LIN {X 0,Y 115.59,Z 711.815,A -85,B 0,C 180,E1 -30048.636,E2 -30048.636} C_VEL
LIN {X 0,Y 121.529,Z 700.022,A -85,B 0,C 180,E1 -30049.447,E2 -30049.447} C_VEL
LIN {X 0,Y 126.039,Z 688.294,A -85,B 0,C 180,E1 -30050.037,E2 -30050.037} C_VEL
LIN {X 0,Y 129.547,Z 675.475,A -85,B 0,C 180,E1 -30050.461,E2 -30050.461} C_VEL
LIN {X 0,Y 131.84,Z 661.062,A -85,B 0,C 180,E1 -30050.822,E2 -30050.822} C_VEL
LIN {X 0,Y 132.217,Z 657.756,A -85,B 0,C 180,E1 -30050.921,E2 -30050.921} C_VEL
LIN {X 0,Y 131.722,Z 655.629,A -85,B 0,C 180,E1 -30053.683,E2 -30053.683} C_VEL
LIN {X 0,Y 131.497,Z 654.069,A -85,B 0,C 180,E1 -30056.17,E2 -30056.17} C_VEL
LIN {X 0,Y 131.404,Z 653.558,A -85,B 0,C 180,E1 -30060.001,E2 -30060.001} C_VEL
LIN {X 0,Y 131.546,Z 654.495,A -85,B 0,C 180,E1 -30062.788,E2 -30062.788} C_VEL
LIN {X 0,Y 131.537,Z 656.009,A -85,B 0,C 180,E1 -30063.787,E2 -30063.787} C_VEL
LIN {X 0,Y 131.334,Z 659.04,A -85,B 0,C 180,E1 -30064.554,E2 -30064.554} C_VEL
LIN {X 0,Y 130.805,Z 663.674,A -85,B 0,C 180,E1 -30064.929,E2 -30064.929} C_VEL
LIN {X 0,Y 129.936,Z 669.022,A -85,B 0,C 180,E1 -30064.793,E2 -30064.793} C_VEL
LIN {X 0,Y 128.707,Z 675.107,A -85,B 0,C 180,E1 -30064.796,E2 -30064.796} C_VEL
LIN {X 0,Y 125.026,Z 688.126,A -85,B 0,C 180,E1 -30065.242,E2 -30065.242} C_VEL
LIN {X 0,Y 120.094,Z 700.491,A -85,B 0,C 180,E1 -30065.831,E2 -30065.831} C_VEL
LIN {X 0,Y 114.09,Z 711.929,A -85,B 0,C 180,E1 -30066.646,E2 -30066.646} C_VEL
LIN {X 0,Y 106.425,Z 723.397,A -85,B 0,C 180,E1 -30067.891,E2 -30067.891} C_VEL
LIN {X 0,Y 97.926,Z 733.578,A -85,B 0,C 180,E1 -30069.321,E2 -30069.321} C_VEL
LIN {X 0,Y 89.47,Z 741.809,A -85,B 0,C 180,E1 -30070.928,E2 -30070.928} C_VEL
LIN {X 0,Y 79.475,Z 749.839,A -85,B 0,C 180,E1 -30073.417,E2 -30073.417} C_VEL
LIN {X 0,Y 69.638,Z 756.292,A -85,B 0,C 180,E1 -30076.516,E2 -30076.516} C_VEL
LIN {X 0,Y 60.109,Z 761.402,A -85,B 0,C 180,E1 -30080.716,E2 -30080.716} C_VEL
LIN {X 0,Y 51.033,Z 765.333,A -85,B 0,C 180,E1 -30086.475,E2 -30086.475} C_VEL
LIN {X 0,Y 42.512,Z 768.222,A -85,B 0,C 180,E1 -30094.253,E2 -30094.253} C_VEL
LIN {X 0,Y 33.116,Z 770.553,A -85,B 0,C 180,E1 -30110.457,E2 -30110.457} C_VEL
LIN {X 0,Y 29.749,Z 771.131,A -85,B 0,C 180,E1 -30121.805,E2 -30121.805} C_VEL
LIN {X 0,Y 27.663,Z 771.312,A -85,B 0,C 180,E1 -30135.283,E2 -30135.283} C_VEL
LIN {X 0,Y 27.148,Z 771.065,A -85,B 0,C 180,E1 -30150,E2 -30150} C_VEL
LIN {X 0,Y 28.19,Z 770.44,A -85,B 0,C 180,E1 -30164.436,E2 -30164.436} C_VEL
LIN {X 0,Y 30.59,Z 769.436,A -85,B 0,C 180,E1 -30177.354,E2 -30177.354} C_VEL
LIN {X 0,Y 34.116,Z 768.006,A -85,B 0,C 180,E1 -30188.17,E2 -30188.17} C_VEL
LIN {X 0,Y 41.107,Z 765.059,A -85,B 0,C 180,E1 -30200.294,E2 -30200.294} C_VEL
LIN {X 0,Y 46.719,Z 762.376,A -85,B 0,C 180,E1 -30206.52,E2 -30206.52} C_VEL
LIN {X 0,Y 46.259,Z 762.112,A -85,B 0,C 180,E1 -30209.388,E2 -30209.388} C_VEL
LIN {X 0,Y 44.988,Z 762.224,A -85,B 0,C 180,E1 -30212.05,E2 -30212.05} C_VEL
LIN {X 0,Y 42.91,Z 762.139,A -85,B 0,C 180,E1 -30220.876,E2 -30220.876} C_VEL
LIN {X 0,Y 41.474,Z 762.242,A -85,B 0,C 180,E1 -30230.242,E2 -30230.242} C_VEL
LIN {X 0,Y 45.335,Z 762.004,A -85,B 0,C 180,E1 -30258.06,E2 -30258.06} C_VEL
LIN {X 0,Y 48.651,Z 761.909,A -85,B 0,C 180,E1 -30265.68,E2 -30265.68} C_VEL
LIN {X 0,Y 47.899,Z 762.718,A -85,B 0,C 180,E1 -30268.318,E2 -30268.318} C_VEL
LIN {X 0,Y 39.67,Z 766.691,A -85,B 0,C 180,E1 -30277.135,E2 -30277.135} C_VEL
LIN {X 0,Y 32.833,Z 769.618,A -85,B 0,C 180,E1 -30290.048,E2 -30290.048} C_VEL
LIN {X 0,Y 29.517,Z 771.007,A -85,B 0,C 180,E1 -30301.563,E2 -30301.563} C_VEL
LIN {X 0,Y 27.544,Z 771.994,A -85,B 0,C 180,E1 -30315.217,E2 -30315.217} C_VEL
LIN {X 0,Y 27.126,Z 772.588,A -85,B 0,C 180,E1 -30330,E2 -30330} C_VEL
LIN {X 0,Y 27.557,Z 772.746,A -85,B 0,C 180,E1 -30344.775,E2 -30344.775} C_VEL
LIN {X 0,Y 32.899,Z 771.821,A -85,B 0,C 180,E1 -30369.856,E2 -30369.856} C_VEL
LIN {X 0,Y 37.238,Z 770.778,A -85,B 0,C 180,E1 -30379.017,E2 -30379.017} C_VEL
LIN {X 0,Y 42.388,Z 769.299,A -85,B 0,C 180,E1 -30385.996,E2 -30385.996} C_VEL
LIN {X 0,Y 50.941,Z 766.283,A -85,B 0,C 180,E1 -30393.733,E2 -30393.733} C_VEL
LIN {X 0,Y 62.114,Z 761.207,A -85,B 0,C 180,E1 -30400.159,E2 -30400.159} C_VEL
LIN {X 0,Y 72.994,Z 754.959,A -85,B 0,C 180,E1 -30404.322,E2 -30404.322} C_VEL
LIN {X 0,Y 82.933,Z 747.864,A -85,B 0,C 180,E1 -30407.037,E2 -30407.037} C_VEL
LIN {X 0,Y 93.039,Z 739.053,A -85,B 0,C 180,E1 -30409.105,E2 -30409.105} C_VEL
LIN {X 0,Y 101.542,Z 729.994,A -85,B 0,C 180,E1 -30410.49,E2 -30410.49} C_VEL
LIN {X 0,Y 109.243,Z 719.912,A -85,B 0,C 180,E1 -30411.535,E2 -30411.535} C_VEL
LIN {X 0,Y 116.123,Z 708.762,A -85,B 0,C 180,E1 -30412.319,E2 -30412.319} C_VEL
LIN {X 0,Y 121.57,Z 697.557,A -85,B 0,C 180,E1 -30412.908,E2 -30412.908} C_VEL
LIN {X 0,Y 126.04,Z 685.303,A -85,B 0,C 180,E1 -30413.325,E2 -30413.325} C_VEL
LIN {X 0,Y 129.305,Z 672.284,A -85,B 0,C 180,E1 -30413.636,E2 -30413.636} C_VEL
LIN {X 0,Y 130.784,Z 662.762,A -85,B 0,C 180,E1 -30413.928,E2 -30413.928} C_VEL
LIN {X 0,Y 130.572,Z 660.969,A -85,B 0,C 180,E1 -30416.915,E2 -30416.915} C_VEL
LIN {X 0,Y 130.533,Z 660.648,A -85,B 0,C 180,E1 -30420.001,E2 -30420.001} C_VEL
LIN {X 0,Y 130.622,Z 661.461,A -85,B 0,C 180,E1 -30422.313,E2 -30422.313} C_VEL
LIN {X 0,Y 130.818,Z 662.851,A -85,B 0,C 180,E1 -30424.506,E2 -30424.506} C_VEL
LIN {X 0,Y 128.707,Z 675.107,A -85,B 0,C 180,E1 -30424.796,E2 -30424.796} C_VEL
LIN {X 0,Y 127.276,Z 680.841,A -85,B 0,C 180,E1 -30424.597,E2 -30424.597} C_VEL
LIN {X 0,Y 124.145,Z 690.015,A -85,B 0,C 180,E1 -30423.615,E2 -30423.615} C_VEL
LIN {X 0,Y 120.303,Z 698.922,A -85,B 0,C 180,E1 -30422.7,E2 -30422.7} C_VEL
LIN {X 0,Y 117.718,Z 704.215,A -85,B 0,C 180,E1 -30422.644,E2 -30422.644} C_VEL
LIN {X 0,Y 111.05,Z 715.823,A -85,B 0,C 180,E1 -30423.361,E2 -30423.361} C_VEL
LIN {X 0,Y 103.089,Z 726.716,A -85,B 0,C 180,E1 -30424.425,E2 -30424.425} C_VEL
LIN {X 0,Y 93.572,Z 737.144,A -85,B 0,C 180,E1 -30425.641,E2 -30425.641} C_VEL
LIN {X 0,Y 84.967,Z 744.801,A -85,B 0,C 180,E1 -30426.999,E2 -30426.999} C_VEL
LIN {X 0,Y 74.727,Z 752.258,A -85,B 0,C 180,E1 -30429.071,E2 -30429.071} C_VEL
LIN {X 0,Y 64.603,Z 758.242,A -85,B 0,C 180,E1 -30431.743,E2 -30431.743} C_VEL
LIN {X 0,Y 54.708,Z 762.953,A -85,B 0,C 180,E1 -30435.539,E2 -30435.539} C_VEL
LIN {X 0,Y 45.124,Z 766.538,A -85,B 0,C 180,E1 -30440.857,E2 -30440.857} C_VEL
LIN {X 0,Y 38.955,Z 768.384,A -85,B 0,C 180,E1 -30445.573,E2 -30445.573} C_VEL
LIN {X 0,Y 33.169,Z 769.762,A -85,B 0,C 180,E1 -30452.056,E2 -30452.056} C_VEL
LIN {X 0,Y 23.716,Z 771.314,A -85,B 0,C 180,E1 -30473.654,E2 -30473.654} C_VEL
LIN {X 0,Y 20.883,Z 771.504,A -85,B 0,C 180,E1 -30490.335,E2 -30490.335} C_VEL
LIN {X 0,Y 20.042,Z 771.264,A -85,B 0,C 180,E1 -30510,E2 -30510} C_VEL
LIN {X 0,Y 21.406,Z 770.644,A -85,B 0,C 180,E1 -30529.166,E2 -30529.166} C_VEL
LIN {X 0,Y 24.5,Z 769.646,A -85,B 0,C 180,E1 -30545.008,E2 -30545.008} C_VEL
LIN {X 0,Y 28.875,Z 768.227,A -85,B 0,C 180,E1 -30556.899,E2 -30556.899} C_VEL
LIN {X 0,Y 38.008,Z 764.859,A -85,B 0,C 180,E1 -30569.88,E2 -30569.88} C_VEL
LIN {X 0,Y 37.473,Z 764.693,A -85,B 0,C 180,E1 -30573.661,E2 -30573.661} C_VEL
LIN {X 0,Y 36.261,Z 764.773,A -85,B 0,C 180,E1 -30611.173,E2 -30611.173} C_VEL
LIN {X 0,Y 39.092,Z 764.687,A -85,B 0,C 180,E1 -30621.071,E2 -30621.071} C_VEL
LIN {X 0,Y 38.792,Z 765.232,A -85,B 0,C 180,E1 -30625.063,E2 -30625.063} C_VEL
LIN {X 0,Y 32.944,Z 767.529,A -85,B 0,C 180,E1 -30631.427,E2 -30631.427} C_VEL
LIN {X 0,Y 27.745,Z 769.399,A -85,B 0,C 180,E1 -30640.545,E2 -30640.545} C_VEL
LIN {X 0,Y 23.494,Z 770.797,A -85,B 0,C 180,E1 -30653.254,E2 -30653.254} C_VEL
LIN {X 0,Y 20.748,Z 771.789,A -85,B 0,C 180,E1 -30670.201,E2 -30670.201} C_VEL
LIN {X 0,Y 20.018,Z 772.388,A -85,B 0,C 180,E1 -30690,E2 -30690} C_VEL
LIN {X 0,Y 20.761,Z 772.557,A -85,B 0,C 180,E1 -30709.786,E2 -30709.786} C_VEL
LIN {X 0,Y 27.799,Z 771.643,A -85,B 0,C 180,E1 -30739.325,E2 -30739.325} C_VEL
LIN {X 0,Y 33.001,Z 770.606,A -85,B 0,C 180,E1 -30748.411,E2 -30748.411} C_VEL
LIN {X 0,Y 38.851,Z 769.138,A -85,B 0,C 180,E1 -30754.751,E2 -30754.751} C_VEL
LIN {X 0,Y 48.215,Z 766.135,A -85,B 0,C 180,E1 -30761.342,E2 -30761.342} C_VEL
LIN {X 0,Y 59.314,Z 761.438,A -85,B 0,C 180,E1 -30766.293,E2 -30766.293} C_VEL
LIN {X 0,Y 71.402,Z 754.842,A -85,B 0,C 180,E1 -30769.822,E2 -30769.822} C_VEL
LIN {X 0,Y 81.635,Z 747.768,A -85,B 0,C 180,E1 -30771.899,E2 -30771.899} C_VEL
LIN {X 0,Y 91.96,Z 738.978,A -85,B 0,C 180,E1 -30773.46,E2 -30773.46} C_VEL
LIN {X 0,Y 100.611,Z 729.948,A -85,B 0,C 180,E1 -30774.494,E2 -30774.494} C_VEL
LIN {X 0,Y 108.427,Z 719.906,A -85,B 0,C 180,E1 -30775.239,E2 -30775.239} C_VEL
LIN {X 0,Y 115.389,Z 708.8,A -85,B 0,C 180,E1 -30775.81,E2 -30775.81} C_VEL
LIN {X 0,Y 121.282,Z 696.784,A -85,B 0,C 180,E1 -30776.264,E2 -30776.264} C_VEL
LIN {X 0,Y 125.89,Z 683.969,A -85,B 0,C 180,E1 -30776.556,E2 -30776.556} C_VEL
LIN {X 0,Y 129.144,Z 670.629,A -85,B 0,C 180,E1 -30776.816,E2 -30776.816} C_VEL
LIN {X 0,Y 129.549,Z 668.159,A -85,B 0,C 180,E1 -30776.891,E2 -30776.891} C_VEL
LIN {X 0,Y 129.532,Z 667.718,A -85,B 0,C 180,E1 -30780.001,E2 -30780.001} C_VEL
LIN {X 0,Y 129.541,Z 668.233,A -85,B 0,C 180,E1 -30781.471,E2 -30781.471} C_VEL
LIN {X 0,Y 126.782,Z 680.85,A -85,B 0,C 180,E1 -30781.786,E2 -30781.786} C_VEL
LIN {X 0,Y 122.426,Z 693.772,A -85,B 0,C 180,E1 -30782.194,E2 -30782.194} C_VEL
LIN {X 0,Y 117.718,Z 704.215,A -85,B 0,C 180,E1 -30782.644,E2 -30782.644} C_VEL
LIN {X 0,Y 114.915,Z 709.418,A -85,B 0,C 180,E1 -30782.615,E2 -30782.615} C_VEL
LIN {X 0,Y 109.743,Z 717.691,A -85,B 0,C 180,E1 -30781.745,E2 -30781.745} C_VEL
LIN {X 0,Y 103.924,Z 725.496,A -85,B 0,C 180,E1 -30780.792,E2 -30780.792} C_VEL
LIN {X 0,Y 100.069,Z 729.966,A -85,B 0,C 180,E1 -30780.712,E2 -30780.712} C_VEL
LIN {X 0,Y 91.391,Z 738.842,A -85,B 0,C 180,E1 -30781.447,E2 -30781.447} C_VEL
LIN {X 0,Y 80.906,Z 747.563,A -85,B 0,C 180,E1 -30782.642,E2 -30782.642} C_VEL
LIN {X 0,Y 70.463,Z 754.546,A -85,B 0,C 180,E1 -30784.151,E2 -30784.151} C_VEL
LIN {X 0,Y 60.091,Z 760.088,A -85,B 0,C 180,E1 -30786.227,E2 -30786.227} C_VEL
LIN {X 0,Y 49.838,Z 764.419,A -85,B 0,C 180,E1 -30789.213,E2 -30789.213} C_VEL
LIN {X 0,Y 43.106,Z 766.693,A -85,B 0,C 180,E1 -30791.978,E2 -30791.978} C_VEL
LIN {X 0,Y 36.455,Z 768.545,A -85,B 0,C 180,E1 -30795.443,E2 -30795.443} C_VEL
LIN {X 0,Y 29.997,Z 769.934,A -85,B 0,C 180,E1 -30800.424,E2 -30800.424} C_VEL
LIN {X 0,Y 18.478,Z 771.497,A -85,B 0,C 180,E1 -30820.475,E2 -30820.475} C_VEL
LIN {X 0,Y 14.389,Z 771.696,A -85,B 0,C 180,E1 -30840.764,E2 -30840.764} C_VEL
LIN {X 0,Y 12.951,Z 771.463,A -85,B 0,C 180,E1 -30870,E2 -30870} C_VEL
LIN {X 0,Y 14.894,Z 770.848,A -85,B 0,C 180,E1 -30898.154,E2 -30898.154} C_VEL
LIN {X 0,Y 19.128,Z 769.856,A -85,B 0,C 180,E1 -30917.293,E2 -30917.293} C_VEL
LIN {X 0,Y 28.63,Z 767.264,A -85,B 0,C 180,E1 -30934.382,E2 -30934.382} C_VEL
LIN {X 0,Y 29.039,Z 766.897,A -85,B 0,C 180,E1 -30940.375,E2 -30940.375} C_VEL
LIN {X 0,Y 29.672,Z 766.991,A -85,B 0,C 180,E1 -30973.698,E2 -30973.698} C_VEL
LIN {X 0,Y 29.855,Z 767.302,A -85,B 0,C 180,E1 -30979.678,E2 -30979.678} C_VEL
LIN {X 0,Y 23.727,Z 769.179,A -85,B 0,C 180,E1 -30987.304,E2 -30987.304} C_VEL
LIN {X 0,Y 18.291,Z 770.586,A -85,B 0,C 180,E1 -30999.787,E2 -30999.787} C_VEL
LIN {X 0,Y 14.25,Z 771.584,A -85,B 0,C 180,E1 -31020.451,E2 -31020.451} C_VEL
LIN {X 0,Y 12.924,Z 772.189,A -85,B 0,C 180,E1 -31050,E2 -31050} C_VEL
LIN {X 0,Y 14.262,Z 772.367,A -85,B 0,C 180,E1 -31079.523,E2 -31079.523} C_VEL
LIN {X 0,Y 23.766,Z 771.464,A -85,B 0,C 180,E1 -31112.513,E2 -31112.513} C_VEL
LIN {X 0,Y 29.889,Z 770.433,A -85,B 0,C 180,E1 -31120.137,E2 -31120.137} C_VEL
LIN {X 0,Y 36.386,Z 768.977,A -85,B 0,C 180,E1 -31124.958,E2 -31124.958} C_VEL
LIN {X 0,Y 46.431,Z 765.986,A -85,B 0,C 180,E1 -31129.689,E2 -31129.689} C_VEL
LIN {X 0,Y 57.084,Z 761.748,A -85,B 0,C 180,E1 -31132.93,E2 -31132.93} C_VEL
LIN {X 0,Y 68.755,Z 755.726,A -85,B 0,C 180,E1 -31135.272,E2 -31135.272} C_VEL
LIN {X 0,Y 79.194,Z 748.96,A -85,B 0,C 180,E1 -31136.706,E2 -31136.706} C_VEL
LIN {X 0,Y 89.675,Z 740.506,A -85,B 0,C 180,E1 -31137.728,E2 -31137.728} C_VEL
LIN {X 0,Y 98.427,Z 731.822,A -85,B 0,C 180,E1 -31138.418,E2 -31138.418} C_VEL
LIN {X 0,Y 107.192,Z 721.142,A -85,B 0,C 180,E1 -31138.946,E2 -31138.946} C_VEL
LIN {X 0,Y 112.456,Z 713.291,A -85,B 0,C 180,E1 -31139.225,E2 -31139.225} C_VEL
LIN {X 0,Y 112.449,Z 713.292,A -85,B 0,C 180,E1 -31139.556,E2 -31139.556} C_VEL
LIN {X 0,Y 104.54,Z 724.592,A -85,B 0,C 180,E1 -31140.29,E2 -31140.29} C_VEL
LIN {X 0,Y 100.069,Z 729.966,A -85,B 0,C 180,E1 -31140.712,E2 -31140.712} C_VEL
LIN {X 0,Y 99.544,Z 731.32,A -85,B 0,C 180,E1 -31140.746,E2 -31140.746} C_VEL
LIN {X 0,Y 99.544,Z 772.025,A -85,B 0,C 180,E1 -31140.746,E2 -31140.746} C_VEL
LIN {X 0,Y 59.705,Z 772.025,A -85,B 0,C 180,E1 -31139.693,E2 -31139.693} C_VEL
LIN {X 0,Y 57.707,Z 770.025,A -85,B 0,C 180,E1 -31139.602,E2 -31139.602} C_VEL
LIN {X 0,Y 57.707,Z 764.186,A -85,B 0,C 180,E1 -31139.602,E2 -31139.602} C_VEL
LIN {X 0,Y 55.003,Z 762.325,A -85,B 0,C 180,E1 -31140.002,E2 -31140.002} C_VEL
LIN {X 0,Y 42.205,Z 766.848,A -85,B 0,C 180,E1 -31142.448,E2 -31142.448} C_VEL
LIN {X 0,Y 35.235,Z 768.705,A -85,B 0,C 180,E1 -31144.236,E2 -31144.236} C_VEL
LIN {X 0,Y 28.308,Z 770.107,A -85,B 0,C 180,E1 -31146.765,E2 -31146.765} C_VEL
LIN {X 0,Y 14.873,Z 771.681,A -85,B 0,C 180,E1 -31159.083,E2 -31159.083} C_VEL
LIN {X 0,Y 8.898,Z 771.888,A -85,B 0,C 180,E1 -31177.834,E2 -31177.834} C_VEL
LIN {X 0,Y 5.87,Z 771.662,A -85,B 0,C 180,E1 -31230,E2 -31230} C_VEL
LIN {X 0,Y 9.262,Z 771.053,A -85,B 0,C 180,E1 -31279.355,E2 -31279.355} C_VEL
LIN {X 0,Y 20.134,Z 769.048,A -85,B 0,C 180,E1 -31303.714,E2 -31303.714} C_VEL
LIN {X 0,Y 21.237,Z 768.763,A -85,B 0,C 180,E1 -31313.11,E2 -31313.11} C_VEL
LIN {X 0,Y 21.34,Z 768.778,A -85,B 0,C 180,E1 -31319.996,E2 -31319.996} C_VEL
LIN {X 0,Y 21.412,Z 768.957,A -85,B 0,C 180,E1 -31330.047,E2 -31330.047} C_VEL
LIN {X 0,Y 14.781,Z 770.375,A -85,B 0,C 180,E1 -31338.025,E2 -31338.025} C_VEL
LIN {X 0,Y 8.793,Z 771.379,A -85,B 0,C 180,E1 -31356.94,E2 -31356.94} C_VEL
LIN {X 0,Y 5.818,Z 771.99,A -85,B 0,C 180,E1 -31410,E2 -31410} C_VEL
LIN {X 0,Y 8.801,Z 772.176,A -85,B 0,C 180,E1 -31462.991,E2 -31462.991} C_VEL
LIN {X 0,Y 14.797,Z 771.925,A -85,B 0,C 180,E1 -31481.783,E2 -31481.783} C_VEL
LIN {X 0,Y 28.274,Z 770.261,A -85,B 0,C 180,E1 -31493.848,E2 -31493.848} C_VEL
LIN {X 0,Y 35.216,Z 768.816,A -85,B 0,C 180,E1 -31496.225,E2 -31496.225} C_VEL
LIN {X 0,Y 45.697,Z 765.838,A -85,B 0,C 180,E1 -31498.497,E2 -31498.497} C_VEL
LIN {X 0,Y 55.003,Z 762.325,A -85,B 0,C 180,E1 -31500.002,E2 -31500.002} C_VEL
LIN {X 0,Y 55.003,Z 762.325,A -85,B 0,C 180,E1 -31500.002,E2 -31500.002}

QRS_NEXT_CUT()

QRS_NEXT()
QRS_HOME()

END
